TYPE Rec_Clamp :
	STRUCT
		Release_Instance				:LREAL;
	END_STRUCT
END_TYPE

(* stored: Version 1.1.0.1, ProductVersion 3.1.4020.12
   DUT Rec_Clamp: Id {0818bec9-89ed-4495-ac2f-2f5459091888} *)
